// TIA Portal V16 export
// export: Created 2021-12-01T20:36:15.3314059Z, ExportSetting WithDefaults, DisplayName Totally Integrated Automation Portal, DisplayVersion V16 Update 4, DisplayName TIA Portal Version Control Interface, DisplayVersion V16 Update 2, DisplayName TIA Portal Openness, DisplayVersion V16 Update 4, DisplayName SINAMICS Startdrive Advanced, DisplayVersion V16 Update 5, DisplayName SINAMICS Startdrive G130, G150, S120, S150, SINAMICS MV, S210, DisplayVersion V16 Update 5, DisplayName SINAMICS Startdrive G110M, G120, G120C, G120D, G120P, G115D, DisplayVersion V16 Update 5, DisplayName STEP 7 Professional, DisplayVersion V16 Update 4, DisplayName STEP 7 Safety, DisplayVersion V16, DisplayName WinCC Advanced, DisplayVersion V16 Update 4
FUNCTION "ST00315_FC" : Void   // FC108, LAD
TITLE = ST00315
{ S7_Optimized_Access := 'TRUE' }
VERSION : 0.1
// stored: AutoNumber true, IsIECCheckEnabled false, SetENOAutomatically false, UDAEnableTagReadback false
   VAR_IN_OUT
      OPMODE : "OPMODE_OUT_UDT";
      HMI_EXTENSION : "HMI_EXTENSION_PANEL_UDT";
   END_VAR
   VAR_TEMP
      EmptyHS : "RT_HANDSHAKE_UDT";
      PlantIdentifier : WString;
   END_VAR
   VAR CONSTANT
      SetLocationUID : String := 'ST00315_SL';
   END_VAR
   VAR_TEMP   // added for the SCL form of the ladder/FBD networks
      _w1 : Bool;
      _w2 : Bool;
   END_VAR
BEGIN

REGION Network 1: Alarm
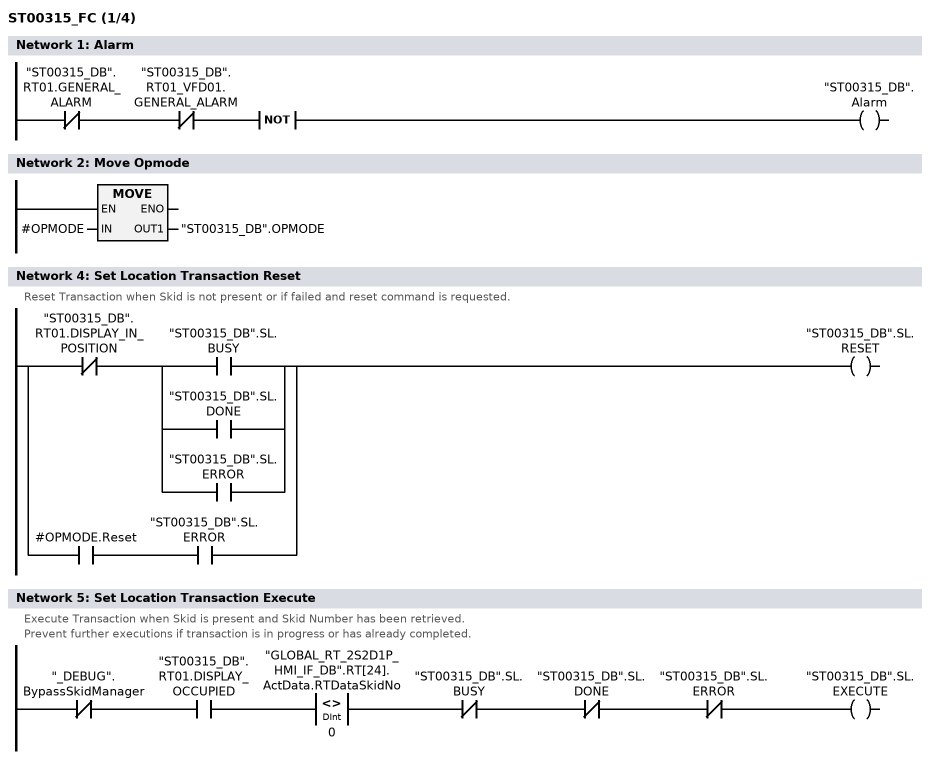
   RUNG wire#powerrail
      I_Contact( "ST00315_DB".RT01.GENERAL_ALARM )
      I_Contact( "ST00315_DB".RT01_VFD01.GENERAL_ALARM )
      Not()
      Coil( "ST00315_DB".Alarm )
   END_RUNG
   // the same network as SCL:
   "ST00315_DB".Alarm := NOT (NOT "ST00315_DB".RT01.GENERAL_ALARM AND NOT "ST00315_DB".RT01_VFD01.GENERAL_ALARM);
END_REGION

REGION Network 2: Move Opmode
   RUNG wire#powerrail
      Move(in := #OPMODE, out1 => "ST00315_DB".OPMODE)
   END_RUNG
   // the same network as SCL:
   "ST00315_DB".OPMODE := #OPMODE;
END_REGION

REGION Network 3: ==== Set Location ====
END_REGION

REGION Network 4: Set Location Transaction Reset
   // Reset Transaction when Skid is not present or if failed and reset command is requested.
   RUNG wire#powerrail
      I_Contact( "ST00315_DB".RT01.DISPLAY_IN_POSITION )
      wire#w1
      Contact( "ST00315_DB".SL.BUSY )
      wire#w2
      Coil( "ST00315_DB".SL.RESET )
   END_RUNG
   RUNG wire#w1
      Contact( "ST00315_DB".SL.DONE )
   END_RUNG wire#w2
   RUNG wire#w1
      Contact( "ST00315_DB".SL.ERROR )
   END_RUNG wire#w2
   RUNG wire#powerrail
      Contact( #OPMODE.Reset )
      Contact( "ST00315_DB".SL.ERROR )
   END_RUNG wire#w2
   // the same network as SCL:
   "ST00315_DB".SL.RESET := (NOT "ST00315_DB".RT01.DISPLAY_IN_POSITION AND ("ST00315_DB".SL.BUSY OR "ST00315_DB".SL.DONE OR "ST00315_DB".SL.ERROR)) OR (#OPMODE.Reset AND "ST00315_DB".SL.ERROR);
END_REGION

REGION Network 5: Set Location Transaction Execute
   // Execute Transaction when Skid is present and Skid Number has been retrieved.
   // Prevent further executions if transaction is in progress or has already completed.
   RUNG wire#powerrail
      I_Contact( "_DEBUG".BypassSkidManager )
      Contact( "ST00315_DB".RT01.DISPLAY_OCCUPIED )
      { S7_Templates := "SrcType := DInt" } NE_Contact(in1 := "GLOBAL_RT_2S2D1P_HMI_IF_DB".RT[24].ActData.RTDataSkidNo, in2 := 0)
      I_Contact( "ST00315_DB".SL.BUSY )
      I_Contact( "ST00315_DB".SL.DONE )
      I_Contact( "ST00315_DB".SL.ERROR )
      Coil( "ST00315_DB".SL.EXECUTE )
   END_RUNG
   // the same network as SCL:
   "ST00315_DB".SL.EXECUTE := NOT "_DEBUG".BypassSkidManager AND "ST00315_DB".RT01.DISPLAY_OCCUPIED AND ("GLOBAL_RT_2S2D1P_HMI_IF_DB".RT[24].ActData.RTDataSkidNo <> 0) AND NOT "ST00315_DB".SL.BUSY AND NOT "ST00315_DB".SL.DONE AND NOT "ST00315_DB".SL.ERROR;
END_REGION

REGION Network 6: Set Location Control
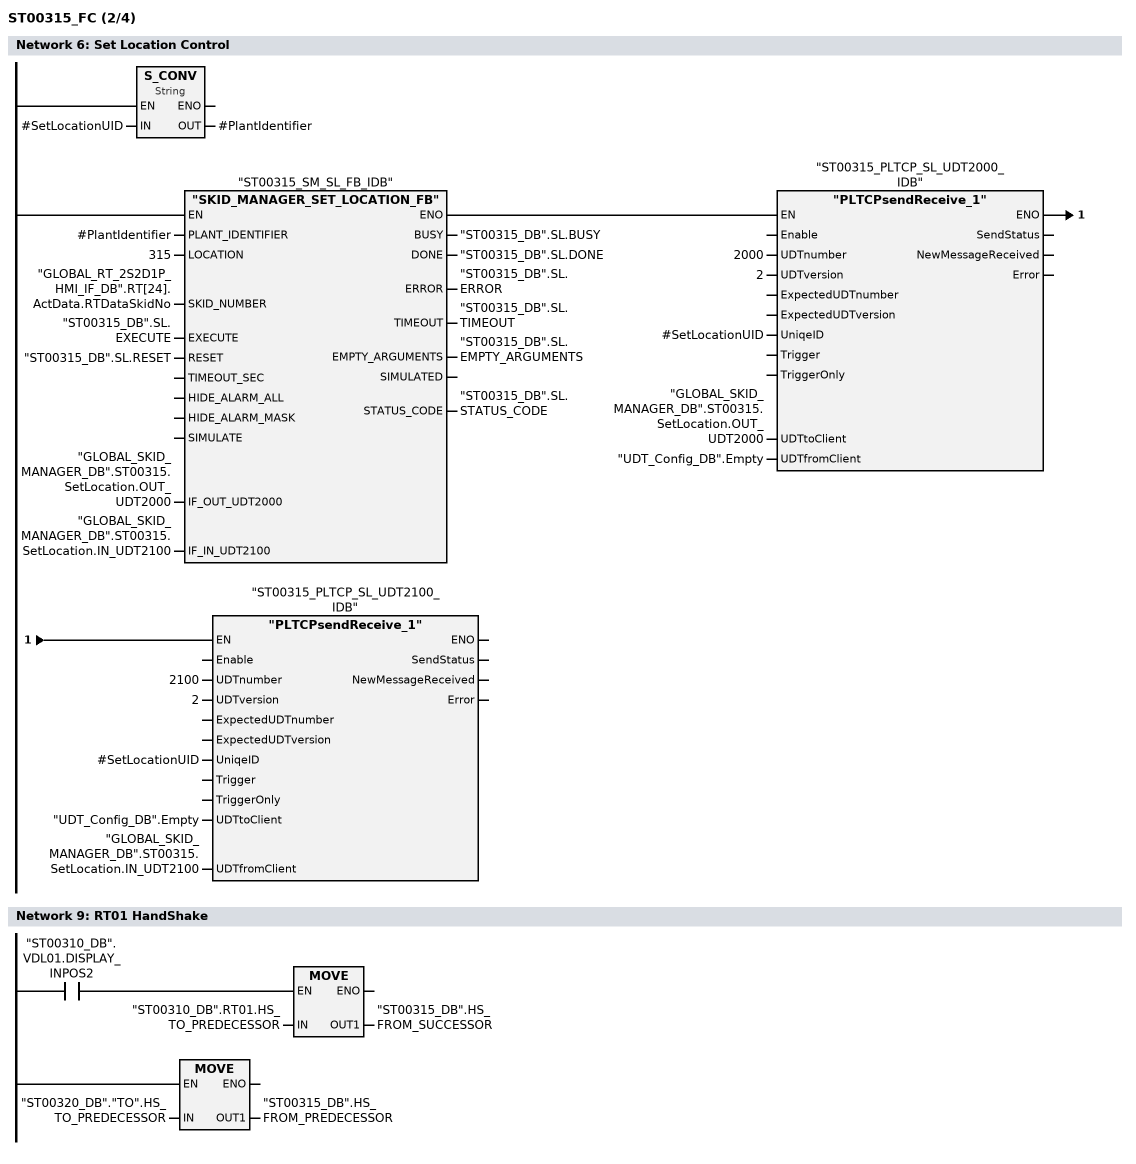
   RUNG wire#powerrail
      { S7_Templates := "[src_type := String, dest_type := WString]" } S_CONV(IN := #SetLocationUID, OUT => #PlantIdentifier)
   END_RUNG
   RUNG wire#powerrail
      "ST00315_SM_SL_FB_IDB"(PLANT_IDENTIFIER := #PlantIdentifier, LOCATION := 315, SKID_NUMBER := "GLOBAL_RT_2S2D1P_HMI_IF_DB".RT[24].ActData.RTDataSkidNo, EXECUTE := "ST00315_DB".SL.EXECUTE, RESET := "ST00315_DB".SL.RESET, TIMEOUT_SEC :=, HIDE_ALARM_ALL :=, HIDE_ALARM_MASK :=, SIMULATE :=, IF_OUT_UDT2000 := "GLOBAL_SKID_MANAGER_DB".ST00315.SetLocation.OUT_UDT2000, IF_IN_UDT2100 := "GLOBAL_SKID_MANAGER_DB".ST00315.SetLocation.IN_UDT2100, BUSY => "ST00315_DB".SL.BUSY, DONE => "ST00315_DB".SL.DONE, ERROR => "ST00315_DB".SL.ERROR, TIMEOUT => "ST00315_DB".SL.TIMEOUT, EMPTY_ARGUMENTS => "ST00315_DB".SL.EMPTY_ARGUMENTS, SIMULATED =>, STATUS_CODE => "ST00315_DB".SL.STATUS_CODE)
      "ST00315_PLTCP_SL_UDT2000_IDB"(Enable :=, UDTnumber := 2000, UDTversion := 2, ExpectedUDTnumber :=, ExpectedUDTversion :=, UniqeID := #SetLocationUID, Trigger :=, TriggerOnly :=, UDTtoClient := "GLOBAL_SKID_MANAGER_DB".ST00315.SetLocation.OUT_UDT2000, UDTfromClient := "UDT_Config_DB".Empty, SendStatus =>, NewMessageReceived =>, Error =>)
      "ST00315_PLTCP_SL_UDT2100_IDB"(Enable :=, UDTnumber := 2100, UDTversion := 2, ExpectedUDTnumber :=, ExpectedUDTversion :=, UniqeID := #SetLocationUID, Trigger :=, TriggerOnly :=, UDTtoClient := "UDT_Config_DB".Empty, UDTfromClient := "GLOBAL_SKID_MANAGER_DB".ST00315.SetLocation.IN_UDT2100, SendStatus =>, NewMessageReceived =>, Error =>)
   END_RUNG
   // the same network as SCL:
   S_CONV(IN := #SetLocationUID, OUT => #PlantIdentifier);
   "ST00315_SM_SL_FB_IDB"(PLANT_IDENTIFIER := #PlantIdentifier,   // "SKID_MANAGER_SET_LOCATION_FB"
                          LOCATION := 315,
                          SKID_NUMBER := "GLOBAL_RT_2S2D1P_HMI_IF_DB".RT[24].ActData.RTDataSkidNo,
                          EXECUTE := "ST00315_DB".SL.EXECUTE,
                          RESET := "ST00315_DB".SL.RESET,
                          IF_OUT_UDT2000 := "GLOBAL_SKID_MANAGER_DB".ST00315.SetLocation.OUT_UDT2000,
                          IF_IN_UDT2100 := "GLOBAL_SKID_MANAGER_DB".ST00315.SetLocation.IN_UDT2100,
                          BUSY => "ST00315_DB".SL.BUSY,
                          DONE => "ST00315_DB".SL.DONE,
                          ERROR => "ST00315_DB".SL.ERROR,
                          TIMEOUT => "ST00315_DB".SL.TIMEOUT,
                          EMPTY_ARGUMENTS => "ST00315_DB".SL.EMPTY_ARGUMENTS,
                          STATUS_CODE => "ST00315_DB".SL.STATUS_CODE,
                          ENO => #_w1);
   "ST00315_PLTCP_SL_UDT2000_IDB"(EN := #_w1,   // "PLTCPsendReceive_1"
                           UDTnumber := 2000,
                           UDTversion := 2,
                           UniqeID := #SetLocationUID,
                           UDTtoClient := "GLOBAL_SKID_MANAGER_DB".ST00315.SetLocation.OUT_UDT2000,
                           UDTfromClient := "UDT_Config_DB".Empty,
                           ENO => #_w2);
   IF #_w2 THEN
       "ST00315_PLTCP_SL_UDT2100_IDB"(UDTnumber := 2100,   // "PLTCPsendReceive_1"
                               UDTversion := 2,
                               UniqeID := #SetLocationUID,
                               UDTtoClient := "UDT_Config_DB".Empty,
                               UDTfromClient := "GLOBAL_SKID_MANAGER_DB".ST00315.SetLocation.IN_UDT2100);
   END_IF;
END_REGION

REGION Network 7: *******************RT01 Control*******************
END_REGION

REGION Network 8 (SCL): RT01 Parameters
   "ST00315_DB".RT01.PARA_SET.Para.PosEndForward1 := true;
   "ST00315_DB".RT01.PARA_SET.Para.PosEndReverse := true;
   "ST00315_DB".RT01.PARA_SET.Para.PosSlowForward := FALSE;
   "ST00315_DB".RT01.PARA_SET.Para.PosSlowReverse := true;
   "ST00315_DB".RT01.PARA_SET.Para.NoStopTrans := true;
   "ST00315_DB".RT01.PARA_SET.Set.RunTimeForward := 450;
   "ST00315_DB".RT01.PARA_SET.Set.RunTimeReverse := 450;
END_REGION

REGION Network 9: RT01 HandShake
   RUNG wire#powerrail
      Contact( "ST00310_DB".VDL01.DISPLAY_INPOS2 )
      Move(in := "ST00310_DB".RT01.HS_TO_PREDECESSOR, out1 => "ST00315_DB".HS_FROM_SUCCESSOR)
   END_RUNG
   RUNG wire#powerrail
      Move(in := "ST00320_DB"."TO".HS_TO_PREDECESSOR, out1 => "ST00315_DB".HS_FROM_PREDECESSOR)
   END_RUNG
   // the same network as SCL:
   IF "ST00310_DB".VDL01.DISPLAY_INPOS2 THEN
       "ST00315_DB".HS_FROM_SUCCESSOR := "ST00310_DB".RT01.HS_TO_PREDECESSOR;
   END_IF;
   "ST00315_DB".HS_FROM_PREDECESSOR := "ST00320_DB"."TO".HS_TO_PREDECESSOR;
END_REGION

REGION Network 10: RT01 FB Control
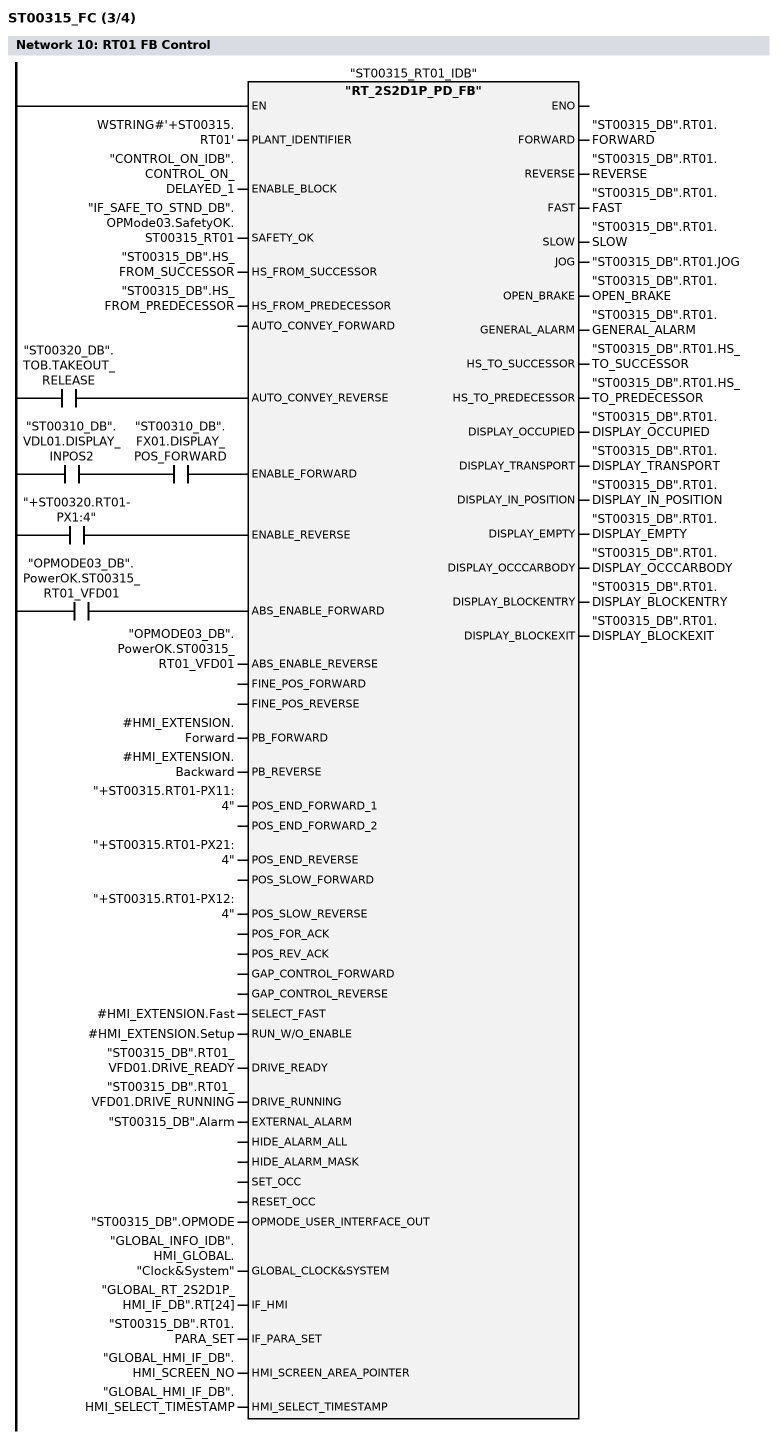
   RUNG wire#powerrail
      "ST00315_RT01_IDB"(AUTO_CONVEY_REVERSE := wire#w1, ENABLE_FORWARD := wire#w2, ENABLE_REVERSE := wire#w3, ABS_ENABLE_FORWARD := wire#w4, PLANT_IDENTIFIER := WSTRING#'+ST00315.RT01', ENABLE_BLOCK := "CONTROL_ON_IDB".CONTROL_ON_DELAYED_1, SAFETY_OK := "IF_SAFE_TO_STND_DB".OPMode03.SafetyOK.ST00315_RT01, HS_FROM_SUCCESSOR := "ST00315_DB".HS_FROM_SUCCESSOR, HS_FROM_PREDECESSOR := "ST00315_DB".HS_FROM_PREDECESSOR, AUTO_CONVEY_FORWARD :=, ABS_ENABLE_REVERSE := "OPMODE03_DB".PowerOK.ST00315_RT01_VFD01, FINE_POS_FORWARD :=, FINE_POS_REVERSE :=, PB_FORWARD := #HMI_EXTENSION.Forward, PB_REVERSE := #HMI_EXTENSION.Backward, POS_END_FORWARD_1 := "+ST00315.RT01-PX11:4", POS_END_FORWARD_2 :=, POS_END_REVERSE := "+ST00315.RT01-PX21:4", POS_SLOW_FORWARD :=, POS_SLOW_REVERSE := "+ST00315.RT01-PX12:4", POS_FOR_ACK :=, POS_REV_ACK :=, GAP_CONTROL_FORWARD :=, GAP_CONTROL_REVERSE :=, SELECT_FAST := #HMI_EXTENSION.Fast, "RUN_W/O_ENABLE" := #HMI_EXTENSION.Setup, DRIVE_READY := "ST00315_DB".RT01_VFD01.DRIVE_READY, DRIVE_RUNNING := "ST00315_DB".RT01_VFD01.DRIVE_RUNNING, EXTERNAL_ALARM := "ST00315_DB".Alarm, HIDE_ALARM_ALL :=, HIDE_ALARM_MASK :=, SET_OCC :=, RESET_OCC :=, OPMODE_USER_INTERFACE_OUT := "ST00315_DB".OPMODE, "GLOBAL_CLOCK&SYSTEM" := "GLOBAL_INFO_IDB".HMI_GLOBAL."Clock&System", IF_HMI := "GLOBAL_RT_2S2D1P_HMI_IF_DB".RT[24], IF_PARA_SET := "ST00315_DB".RT01.PARA_SET, HMI_SCREEN_AREA_POINTER := "GLOBAL_HMI_IF_DB".HMI_SCREEN_NO, HMI_SELECT_TIMESTAMP := "GLOBAL_HMI_IF_DB".HMI_SELECT_TIMESTAMP, FORWARD => "ST00315_DB".RT01.FORWARD, REVERSE => "ST00315_DB".RT01.REVERSE, FAST => "ST00315_DB".RT01.FAST, SLOW => "ST00315_DB".RT01.SLOW, JOG => "ST00315_DB".RT01.JOG, OPEN_BRAKE => "ST00315_DB".RT01.OPEN_BRAKE, GENERAL_ALARM => "ST00315_DB".RT01.GENERAL_ALARM, HS_TO_SUCCESSOR => "ST00315_DB".RT01.HS_TO_SUCCESSOR, HS_TO_PREDECESSOR => "ST00315_DB".RT01.HS_TO_PREDECESSOR, DISPLAY_OCCUPIED => "ST00315_DB".RT01.DISPLAY_OCCUPIED, DISPLAY_TRANSPORT => "ST00315_DB".RT01.DISPLAY_TRANSPORT, DISPLAY_IN_POSITION => "ST00315_DB".RT01.DISPLAY_IN_POSITION, DISPLAY_EMPTY => "ST00315_DB".RT01.DISPLAY_EMPTY, DISPLAY_OCCCARBODY => "ST00315_DB".RT01.DISPLAY_OCCCARBODY, DISPLAY_BLOCKENTRY => "ST00315_DB".RT01.DISPLAY_BLOCKENTRY, DISPLAY_BLOCKEXIT => "ST00315_DB".RT01.DISPLAY_BLOCKEXIT)
   END_RUNG
   RUNG wire#powerrail
      Contact( "ST00320_DB".TOB.TAKEOUT_RELEASE )
   END_RUNG wire#w1
   RUNG wire#powerrail
      Contact( "ST00310_DB".VDL01.DISPLAY_INPOS2 )
      Contact( "ST00310_DB".FX01.DISPLAY_POS_FORWARD )
   END_RUNG wire#w2
   RUNG wire#powerrail
      Contact( "+ST00320.RT01-PX1:4" )
   END_RUNG wire#w3
   RUNG wire#powerrail
      Contact( "OPMODE03_DB".PowerOK.ST00315_RT01_VFD01 )
   END_RUNG wire#w4
   // the same network as SCL:
   "ST00315_RT01_IDB"(PLANT_IDENTIFIER := WSTRING#'+ST00315.RT01',   // "RT_2S2D1P_PD_FB"
                      ENABLE_BLOCK := "CONTROL_ON_IDB".CONTROL_ON_DELAYED_1,
                      SAFETY_OK := "IF_SAFE_TO_STND_DB".OPMode03.SafetyOK.ST00315_RT01,
                      HS_FROM_SUCCESSOR := "ST00315_DB".HS_FROM_SUCCESSOR,
                      HS_FROM_PREDECESSOR := "ST00315_DB".HS_FROM_PREDECESSOR,
                      AUTO_CONVEY_REVERSE := "ST00320_DB".TOB.TAKEOUT_RELEASE,
                      ENABLE_FORWARD := "ST00310_DB".VDL01.DISPLAY_INPOS2 AND "ST00310_DB".FX01.DISPLAY_POS_FORWARD,
                      ENABLE_REVERSE := "+ST00320.RT01-PX1:4",
                      ABS_ENABLE_FORWARD := "OPMODE03_DB".PowerOK.ST00315_RT01_VFD01,
                      ABS_ENABLE_REVERSE := "OPMODE03_DB".PowerOK.ST00315_RT01_VFD01,
                      PB_FORWARD := #HMI_EXTENSION.Forward,
                      PB_REVERSE := #HMI_EXTENSION.Backward,
                      POS_END_FORWARD_1 := "+ST00315.RT01-PX11:4",
                      POS_END_REVERSE := "+ST00315.RT01-PX21:4",
                      POS_SLOW_REVERSE := "+ST00315.RT01-PX12:4",
                      SELECT_FAST := #HMI_EXTENSION.Fast,
                      "RUN_W/O_ENABLE" := #HMI_EXTENSION.Setup,
                      DRIVE_READY := "ST00315_DB".RT01_VFD01.DRIVE_READY,
                      DRIVE_RUNNING := "ST00315_DB".RT01_VFD01.DRIVE_RUNNING,
                      EXTERNAL_ALARM := "ST00315_DB".Alarm,
                      OPMODE_USER_INTERFACE_OUT := "ST00315_DB".OPMODE,
                      "GLOBAL_CLOCK&SYSTEM" := "GLOBAL_INFO_IDB".HMI_GLOBAL."Clock&System",
                      IF_HMI := "GLOBAL_RT_2S2D1P_HMI_IF_DB".RT[24],
                      IF_PARA_SET := "ST00315_DB".RT01.PARA_SET,
                      HMI_SCREEN_AREA_POINTER := "GLOBAL_HMI_IF_DB".HMI_SCREEN_NO,
                      HMI_SELECT_TIMESTAMP := "GLOBAL_HMI_IF_DB".HMI_SELECT_TIMESTAMP,
                      FORWARD => "ST00315_DB".RT01.FORWARD,
                      REVERSE => "ST00315_DB".RT01.REVERSE,
                      FAST => "ST00315_DB".RT01.FAST,
                      SLOW => "ST00315_DB".RT01.SLOW,
                      JOG => "ST00315_DB".RT01.JOG,
                      OPEN_BRAKE => "ST00315_DB".RT01.OPEN_BRAKE,
                      GENERAL_ALARM => "ST00315_DB".RT01.GENERAL_ALARM,
                      HS_TO_SUCCESSOR => "ST00315_DB".RT01.HS_TO_SUCCESSOR,
                      HS_TO_PREDECESSOR => "ST00315_DB".RT01.HS_TO_PREDECESSOR,
                      DISPLAY_OCCUPIED => "ST00315_DB".RT01.DISPLAY_OCCUPIED,
                      DISPLAY_TRANSPORT => "ST00315_DB".RT01.DISPLAY_TRANSPORT,
                      DISPLAY_IN_POSITION => "ST00315_DB".RT01.DISPLAY_IN_POSITION,
                      DISPLAY_EMPTY => "ST00315_DB".RT01.DISPLAY_EMPTY,
                      DISPLAY_OCCCARBODY => "ST00315_DB".RT01.DISPLAY_OCCCARBODY,
                      DISPLAY_BLOCKENTRY => "ST00315_DB".RT01.DISPLAY_BLOCKENTRY,
                      DISPLAY_BLOCKEXIT => "ST00315_DB".RT01.DISPLAY_BLOCKEXIT);
END_REGION

REGION Network 11: RT01 Speed
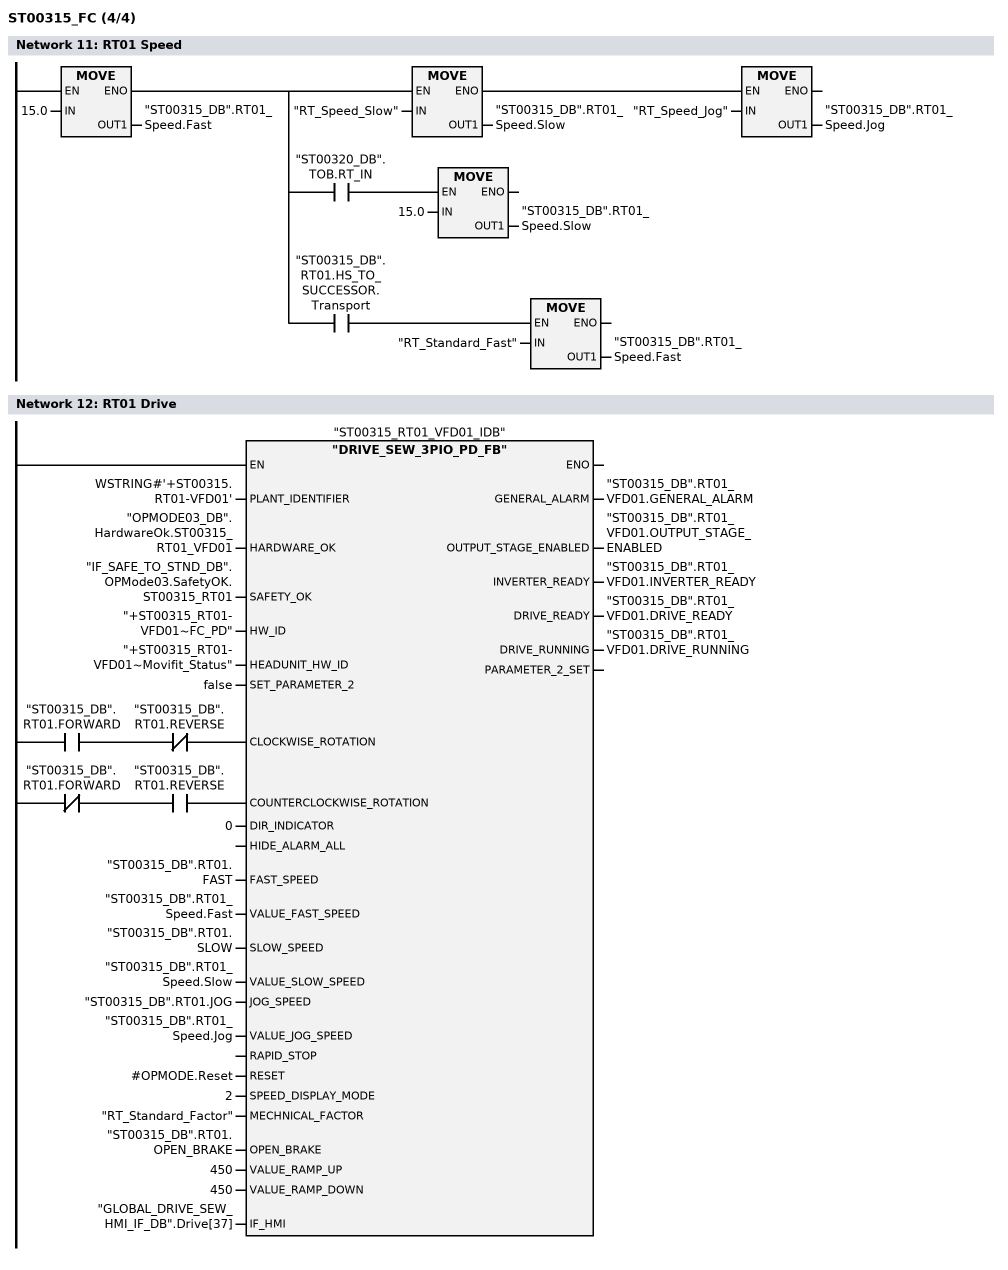
   RUNG wire#powerrail
      Move(in := 15.0, out1 => "ST00315_DB".RT01_Speed.Fast)
      wire#w1
      Move(in := "RT_Speed_Slow", out1 => "ST00315_DB".RT01_Speed.Slow)
      Move(in := "RT_Speed_Jog", out1 => "ST00315_DB".RT01_Speed.Jog)
   END_RUNG
   RUNG wire#w1
      Contact( "ST00320_DB".TOB.RT_IN )
      Move(in := 15.0, out1 => "ST00315_DB".RT01_Speed.Slow)
   END_RUNG
   RUNG wire#w1
      Contact( "ST00315_DB".RT01.HS_TO_SUCCESSOR.Transport )
      Move(in := "RT_Standard_Fast", out1 => "ST00315_DB".RT01_Speed.Fast)
   END_RUNG
   // the same network as SCL:
   "ST00315_DB".RT01_Speed.Fast := 15.0;
   "ST00315_DB".RT01_Speed.Slow := "RT_Speed_Slow";
   "ST00315_DB".RT01_Speed.Jog := "RT_Speed_Jog";
   IF "ST00320_DB".TOB.RT_IN THEN "ST00315_DB".RT01_Speed.Slow := 15.0; END_IF;
   IF "ST00315_DB".RT01.HS_TO_SUCCESSOR.Transport THEN
       "ST00315_DB".RT01_Speed.Fast := "RT_Standard_Fast";
   END_IF;
END_REGION

REGION Network 12: RT01 Drive
   RUNG wire#powerrail
      "ST00315_RT01_VFD01_IDB"(CLOCKWISE_ROTATION := wire#w1, COUNTERCLOCKWISE_ROTATION := wire#w2, PLANT_IDENTIFIER := WSTRING#'+ST00315.RT01-VFD01', HARDWARE_OK := "OPMODE03_DB".HardwareOk.ST00315_RT01_VFD01, SAFETY_OK := "IF_SAFE_TO_STND_DB".OPMode03.SafetyOK.ST00315_RT01, HW_ID := "+ST00315_RT01-VFD01~FC_PD", HEADUNIT_HW_ID := "+ST00315_RT01-VFD01~Movifit_Status", SET_PARAMETER_2 := false, DIR_INDICATOR := 0, HIDE_ALARM_ALL :=, FAST_SPEED := "ST00315_DB".RT01.FAST, VALUE_FAST_SPEED := "ST00315_DB".RT01_Speed.Fast, SLOW_SPEED := "ST00315_DB".RT01.SLOW, VALUE_SLOW_SPEED := "ST00315_DB".RT01_Speed.Slow, JOG_SPEED := "ST00315_DB".RT01.JOG, VALUE_JOG_SPEED := "ST00315_DB".RT01_Speed.Jog, RAPID_STOP :=, RESET := #OPMODE.Reset, SPEED_DISPLAY_MODE := 2, MECHNICAL_FACTOR := "RT_Standard_Factor", OPEN_BRAKE := "ST00315_DB".RT01.OPEN_BRAKE, VALUE_RAMP_UP := 450, VALUE_RAMP_DOWN := 450, IF_HMI := "GLOBAL_DRIVE_SEW_HMI_IF_DB".Drive[37], GENERAL_ALARM => "ST00315_DB".RT01_VFD01.GENERAL_ALARM, OUTPUT_STAGE_ENABLED => "ST00315_DB".RT01_VFD01.OUTPUT_STAGE_ENABLED, INVERTER_READY => "ST00315_DB".RT01_VFD01.INVERTER_READY, DRIVE_READY => "ST00315_DB".RT01_VFD01.DRIVE_READY, DRIVE_RUNNING => "ST00315_DB".RT01_VFD01.DRIVE_RUNNING, PARAMETER_2_SET =>)
   END_RUNG
   RUNG wire#powerrail
      Contact( "ST00315_DB".RT01.FORWARD )
      I_Contact( "ST00315_DB".RT01.REVERSE )
   END_RUNG wire#w1
   RUNG wire#powerrail
      I_Contact( "ST00315_DB".RT01.FORWARD )
      Contact( "ST00315_DB".RT01.REVERSE )
   END_RUNG wire#w2
   // the same network as SCL:
   "ST00315_RT01_VFD01_IDB"(PLANT_IDENTIFIER := WSTRING#'+ST00315.RT01-VFD01',   // "DRIVE_SEW_3PIO_PD_FB"
                           HARDWARE_OK := "OPMODE03_DB".HardwareOk.ST00315_RT01_VFD01,
                           SAFETY_OK := "IF_SAFE_TO_STND_DB".OPMode03.SafetyOK.ST00315_RT01,
                           HW_ID := "+ST00315_RT01-VFD01~FC_PD",
                           HEADUNIT_HW_ID := "+ST00315_RT01-VFD01~Movifit_Status",
                           SET_PARAMETER_2 := false,
                           CLOCKWISE_ROTATION := "ST00315_DB".RT01.FORWARD AND NOT "ST00315_DB".RT01.REVERSE,
                           COUNTERCLOCKWISE_ROTATION := NOT "ST00315_DB".RT01.FORWARD AND "ST00315_DB".RT01.REVERSE,
                           DIR_INDICATOR := 0,
                           FAST_SPEED := "ST00315_DB".RT01.FAST,
                           VALUE_FAST_SPEED := "ST00315_DB".RT01_Speed.Fast,
                           SLOW_SPEED := "ST00315_DB".RT01.SLOW,
                           VALUE_SLOW_SPEED := "ST00315_DB".RT01_Speed.Slow,
                           JOG_SPEED := "ST00315_DB".RT01.JOG,
                           VALUE_JOG_SPEED := "ST00315_DB".RT01_Speed.Jog,
                           RESET := #OPMODE.Reset,
                           SPEED_DISPLAY_MODE := 2,
                           MECHNICAL_FACTOR := "RT_Standard_Factor",
                           OPEN_BRAKE := "ST00315_DB".RT01.OPEN_BRAKE,
                           VALUE_RAMP_UP := 450,
                           VALUE_RAMP_DOWN := 450,
                           IF_HMI := "GLOBAL_DRIVE_SEW_HMI_IF_DB".Drive[37],
                           GENERAL_ALARM => "ST00315_DB".RT01_VFD01.GENERAL_ALARM,
                           OUTPUT_STAGE_ENABLED => "ST00315_DB".RT01_VFD01.OUTPUT_STAGE_ENABLED,
                           INVERTER_READY => "ST00315_DB".RT01_VFD01.INVERTER_READY,
                           DRIVE_READY => "ST00315_DB".RT01_VFD01.DRIVE_READY,
                           DRIVE_RUNNING => "ST00315_DB".RT01_VFD01.DRIVE_RUNNING);
END_REGION
END_FUNCTION
